{attribute 'GeneratedUsingTerminal: EK1100-0000-0018'}
{attribute addProperty BoxType "EK1100-0000-0018"}
{attribute addProperty Id "Term_2_EL1809EL1809_FD7895E220"}
{attribute addProperty CRC "3085915774"}
{attribute addProperty Size "20"}
TYPE Term_1_EK1100_B7EF567E EXTENDS EK1100_AB5A9467 :
STRUCT
	{attribute addProperty Name "Term_2_EL1809"}
	Term_2_EL1809 : EL1809_FD7895E2;
END_STRUCT
END_TYPE

(* stored: Version 1.2.0.0, ProductVersion 3.1.4024.9
   DUT Term_1_EK1100_B7EF567E: Id {ce616fa5-8d67-4da7-92fa-879c4a0def09} *)
